FUNCTION_BLOCK FB_Observable_LWORD EXTENDS FB_AbstractObservable
VAR
    _nVal:              LWORD;
    _nOldVal:           LWORD;
END_VAR

METHOD FB_init : BOOL
VAR_INPUT
    bInitRetains:       BOOL; // if TRUE, the retain variables are initialized (warm start / cold start)
    bInCopyCode:        BOOL;  // if TRUE, the instance afterwards gets moved into the copy code (online change)
END_VAR
THIS^._nTypeClass := __SYSTEM.TYPE_CLASS.TYPE_LWORD;
END_METHOD

PROPERTY nDataSize : UDINT
GET
nDataSize := SIZEOF(LWORD);
END_GET
END_PROPERTY

PROPERTY nValue64 : LWORD
GET
nValue64 := THIS^._nVal;
END_GET
SET
THIS^._nOldVal := THIS^._nVal;
THIS^._nVal := nValue64;

THIS^.NotifyWithConditions();
END_SET
END_PROPERTY

PROPERTY PROTECTED pData : POINTER TO BYTE
GET
pData := ADR(THIS^._nVal);
END_GET
END_PROPERTY

METHOD  ValueChanged : BOOL
VAR_INPUT
END_VAR
ValueChanged := THIS^._nOldVal <> THIS^._nVal;
END_METHOD

END_FUNCTION_BLOCK

(* stored: Version 1.1.0.1, ProductVersion 3.1.4024.12
   POU FB_Observable_LWORD: Id {5dabbb98-9a3a-0da7-08f0-66a3e96a3a98}, SpecialFunc None
   Method FB_init: Id {7c63da85-50a8-0d8d-092a-fb4ca5f33d1a}
   Property nDataSize: Id {bdde6460-531a-0086-1d5a-a22cfc08266d}
   Get Get: Id {859e6ce4-f128-075d-118d-0067c87d142b}
   Property nValue64: Id {718e8ddf-a6e7-0d69-0175-ea38fc62de76}
   Get Get: Id {07441eb5-fa49-0713-0dc3-94a7a619fcfc}
   Set Set: Id {d32649e7-7f51-069e-2a1e-41da77fa37b2}
   Property pData: Id {013c9a9c-0abb-0796-3fd0-d0969af66495}
   Get Get: Id {b9d411c0-18e2-07ac-2055-c3b2001d65b2}
   Method ValueChanged: Id {79d39161-7a34-0ff4-0714-d9f61ecd989b} *)
